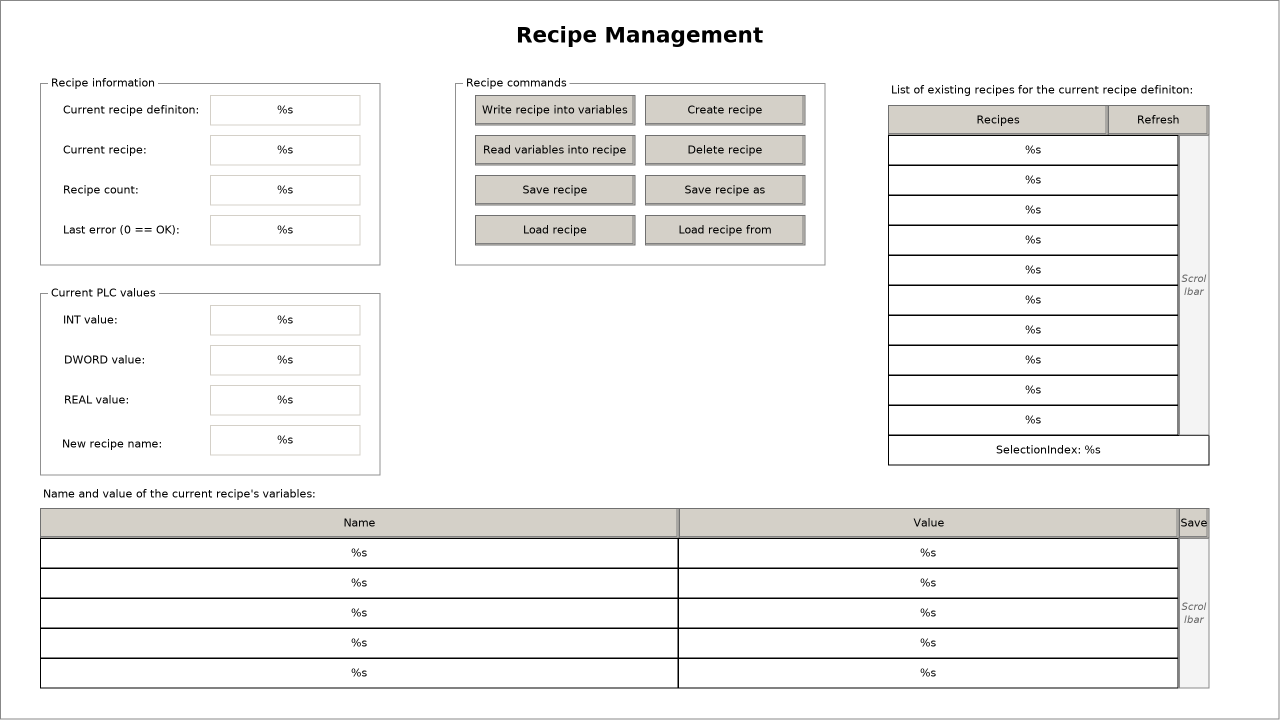
VISUALIZATION Visualization  // 1280x720
    GroupBox (455,75 370x190), "Recipe commands"
        Button (20,20 160x30), "Write recipe into variables"
            OnMouseClick: ExecuteCommand ExecuteCommand=ExecuteCommand=[Command=WriteRecipe, Value=RecipeManagement.sRecipeDef, Value2=RecipeManagement.sRecipe]
        Button (20,60 160x30), "Read variables into recipe"
            OnMouseClick: ExecuteCommand ExecuteCommand=ExecuteCommand=[Command=ReadRecipe, Value=RecipeManagement.sRecipeDef, Value2=RecipeManagement.sRecipe]
            OnMouseClick: execute { RecipeManagement.bReloadValues := TRUE; }
        Button (20,100 160x30), "Save recipe"
            OnMouseClick: ExecuteCommand ExecuteCommand=ExecuteCommand=[Command=SaveRecipe, Value=RecipeManagement.sRecipeDef, Value2=RecipeManagement.sRecipe]
        Button (20,140 160x30), "Load recipe"
            OnMouseClick: ExecuteCommand ExecuteCommand=ExecuteCommand=[Command=LoadRecipe, Value=RecipeManagement.sRecipeDef, Value2=RecipeManagement.sRecipe]
            OnMouseClick: toggle RecipeManagement.bReloadValues
        Button (190,20 160x30), "Create recipe"
            OnMouseClick: ExecuteCommand ExecuteCommand=ExecuteCommand=[Command=CreateRecipe, Value=RecipeManagement.sRecipeDef, Value2=MAIN.sRecipe]
            OnMouseClick: execute { RecipeManagement.bReload := TRUE; }
        Button (190,100 160x30), "Save recipe as"
            OnMouseClick: ExecuteCommand ExecuteCommand=ExecuteCommand=[Command=SaveRecipeAs, Value=RecipeManagement.sRecipeDef, Value2=RecipeManagement.sRecipe]
        Button (190,140 160x30), "Load recipe from"
            OnMouseClick: ExecuteCommand ExecuteCommand=ExecuteCommand=[Command=LoadRecipeFrom, Value=RecipeManagement.sRecipeDef, Value2=RecipeManagement.sRecipe]
        Button (190,60 160x30), "Delete recipe"
            OnMouseClick: ExecuteCommand ExecuteCommand=ExecuteCommand=[Command=DeleteRecipe, Value=RecipeManagement.sRecipeDef, Value2=RecipeManagement.sRecipe]
            OnMouseClick: execute { RecipeManagement.bInit := TRUE; }
    GroupBox (40,285 340x190), "Current PLC values"
        Label (20,20 150x30), "INT value:"
        Textfield (170,20 150x30), "%s", text variable: MAIN.nValueInt
            OnMouseClick: write the text variable via Default
        Label (21,60 150x30), "DWORD value:"
        Textfield (170,60 150x30), "%s", text variable: MAIN.nValueDword
            OnMouseClick: write the text variable via Default
        Label (21,100 150x30), "REAL value:"
        Textfield (170,100 150x30), "%s", text variable: MAIN.fValueReal
            OnMouseClick: write the text variable via Default
        Label (19,144 150x30), "New recipe name:"
        Textfield (170,140 150x30), "%s", text variable: MAIN.sRecipe
            OnMouseClick: write the text variable via Default
    Label (490,20 300x30), "Recipe Management"
    GroupBox (40,75 340x190), "Recipe information"
        Textfield (170,20 150x30), "%s", text variable: RecipeManagement.sRecipeDef
            OnMouseClick: write the text variable via Default
        Label (20,20 150x30), "Current recipe definiton:"
        Label (20,60 150x30), "Current recipe:"
        Label (20,140 150x30), "Last error (0 == OK):"
        Label (20,100 150x30), "Recipe count:"
        Textfield (170,60 150x30), "%s", text variable: RecipeManagement.sRecipe
            OnMouseClick: write the text variable via Default
        Textfield (170,140 150x30), "%s", text variable: RecipeManagement.nLastError
        Textfield (170,100 150x30), "%s", text variable: RecipeManagement.nRecipeCount
    Button (40,508 639x30), "Name"
        OnMouseDown: toggle RecipeManagement.bReload
    Button (679,508 500x30), "Value"
        OnMouseDown: toggle RecipeManagement.bReload
    Rectangle (40,479 305x30), "Name and value of the current recipe's variables:"
    Button (1179,508 30x30), "Save"
        OnMouseDown: toggle RecipeManagement.bSaveVariables
    Rectangle (40,538 638x30), "%s", text variable: GVL_RecipeTable.aVariableNames[0]
    Rectangle (40,568 638x30), "%s", text variable: GVL_RecipeTable.aVariableNames[1]
    Rectangle (40,598 638x30), "%s", text variable: GVL_RecipeTable.aVariableNames[2]
    Rectangle (40,628 638x30), "%s", text variable: GVL_RecipeTable.aVariableNames[3]
    Rectangle (40,658 638x30), "%s", text variable: GVL_RecipeTable.aVariableNames[4]
    Rectangle (678,538 500x30), "%s", text variable: GVL_RecipeTable.aVariableValues[0]
        OnMouseDown: write the text variable via Edit
    Rectangle (678,568 500x30), "%s", text variable: GVL_RecipeTable.aVariableValues[1]
        OnMouseDown: write the text variable via Edit
    Rectangle (678,598 500x30), "%s", text variable: GVL_RecipeTable.aVariableValues[2]
        OnMouseDown: write the text variable via Edit
    Rectangle (678,628 500x30), "%s", text variable: GVL_RecipeTable.aVariableValues[3]
        OnMouseDown: write the text variable via Edit
    Rectangle (678,658 500x30), "%s", text variable: GVL_RecipeTable.aVariableValues[4]
        OnMouseDown: write the text variable via Edit
    Scrollbar (1179,538 30x150)
        p2245068023: GVL_RecipeTable.nRecipeCount
        p1057716461: GVL_RecipeTable.nVariableIndex
    Button (888,105 220x30), "Recipes"
        OnMouseDown: toggle RecipeManagement.bReload
    Label (888,75 322x30), "List of existing recipes for the current recipe definiton:"
    Button (1108,105 101x30), "Refresh"
        OnMouseDown: toggle RecipeManagement.bReload
    Rectangle (888,135 290x30), "%s", text variable: GVL_RecipeTable.aRecipeNames[0], colour toggle: (GVL_RecipeTable.nRecipeSelectionIndex-GVL_RecipeTable.nRecipeIndex) = 0
        OnMouseDown: execute { GVL_RecipeTable.nRecipeSelectionIndex := GVL_RecipeTable.nRecipeIndex; }
    Rectangle (888,165 290x30), "%s", text variable: GVL_RecipeTable.aRecipeNames[1], colour toggle: (GVL_RecipeTable.nRecipeSelectionIndex-GVL_RecipeTable.nRecipeIndex) = 1
        OnMouseDown: execute { GVL_RecipeTable.nRecipeSelectionIndex := GVL_RecipeTable.nRecipeIndex + 1; }
    Rectangle (888,195 290x30), "%s", text variable: GVL_RecipeTable.aRecipeNames[2], colour toggle: (GVL_RecipeTable.nRecipeSelectionIndex-GVL_RecipeTable.nRecipeIndex) = 2
        OnMouseDown: execute { GVL_RecipeTable.nRecipeSelectionIndex := GVL_RecipeTable.nRecipeIndex + 2; }
    Rectangle (888,225 290x30), "%s", text variable: GVL_RecipeTable.aRecipeNames[4], colour toggle: (GVL_RecipeTable.nRecipeSelectionIndex-GVL_RecipeTable.nRecipeIndex) = 3
        OnMouseDown: execute { GVL_RecipeTable.nRecipeSelectionIndex := GVL_RecipeTable.nRecipeIndex + 3; }
    Rectangle (888,255 290x30), "%s", text variable: GVL_RecipeTable.aRecipeNames[5], colour toggle: (GVL_RecipeTable.nRecipeSelectionIndex-GVL_RecipeTable.nRecipeIndex) = 4
        OnMouseDown: execute { GVL_RecipeTable.nRecipeSelectionIndex := GVL_RecipeTable.nRecipeIndex + 4; }
    Rectangle (888,285 290x30), "%s", text variable: GVL_RecipeTable.aRecipeNames[6], colour toggle: (GVL_RecipeTable.nRecipeSelectionIndex-GVL_RecipeTable.nRecipeIndex) = 5
        OnMouseDown: execute { GVL_RecipeTable.nRecipeSelectionIndex := GVL_RecipeTable.nRecipeIndex + 5; }
    Rectangle (888,315 290x30), "%s", text variable: GVL_RecipeTable.aRecipeNames[6], colour toggle: (GVL_RecipeTable.nRecipeSelectionIndex-GVL_RecipeTable.nRecipeIndex) = 6
        OnMouseDown: execute { GVL_RecipeTable.nRecipeSelectionIndex := GVL_RecipeTable.nRecipeIndex + 6; }
    Rectangle (888,345 290x30), "%s", text variable: GVL_RecipeTable.aRecipeNames[7], colour toggle: (GVL_RecipeTable.nRecipeSelectionIndex-GVL_RecipeTable.nRecipeIndex) = 7
        OnMouseDown: execute { GVL_RecipeTable.nRecipeSelectionIndex := GVL_RecipeTable.nRecipeIndex + 7; }
    Rectangle (888,375 290x30), "%s", text variable: GVL_RecipeTable.aRecipeNames[8], colour toggle: (GVL_RecipeTable.nRecipeSelectionIndex-GVL_RecipeTable.nRecipeIndex) = 8
        OnMouseDown: execute { GVL_RecipeTable.nRecipeSelectionIndex := GVL_RecipeTable.nRecipeIndex + 8; }
    Rectangle (888,405 290x30), "%s", text variable: GVL_RecipeTable.aRecipeNames[9], colour toggle: (GVL_RecipeTable.nRecipeSelectionIndex-GVL_RecipeTable.nRecipeIndex) = 9
        OnMouseDown: execute { GVL_RecipeTable.nRecipeSelectionIndex := GVL_RecipeTable.nRecipeIndex + 9; }
    Rectangle (888,435 321x30), "SelectionIndex: %s", text variable: GVL_RecipeTable.nRecipeSelectionIndex+1
    Scrollbar (1179,135 30x300)
        p2245068023: GVL_RecipeTable.nRecipeCount
        p1057716461: GVL_RecipeTable.nRecipeIndex
END_VISUALIZATION

(* stored: Version 1.1.0.1, ProductVersion 3.1.4024.3
   Visu Visualization: Id {7c80b83f-eb0f-4e0e-baee-9070c17c89b8} *)
